// TIA Portal V20 export
// export: Created 2025-12-01T14:56:19.1111183Z, ExportSetting None, DisplayName Totally Integrated Automation Portal, DisplayVersion V20 Update 3, DisplayName TIA Portal Openness, DisplayVersion V20 Update 3, DisplayName TIA Portal Version Control Interface, DisplayVersion V20 Update 3, DisplayName STEP 7 Professional, DisplayVersion V20 Update 3, DisplayName STEP 7 Safety, DisplayVersion V20 Update 2, DisplayName WinCC Basic/Comfort/Advanced, DisplayVersion V20 Update 3, DisplayName WinCC Professional, DisplayVersion V20 Update 3, DisplayName WinCC Unified, DisplayVersion V20 Update 3
TYPE "MOVIMOT_Datos"
   STRUCT
      ENABLE : Bool;
      RESET : Bool;
      BRAKE_RELEASE : Bool;   // without_ENABLE
      "SPEED%" : Int;
      RAMP : Int := 1000;
      READY : Bool;
      FAULT : Bool;
      ERROR_NO : Int;
      CURRENT : Int;
   END_STRUCT;
END_TYPE
